ABB RAPID module: LArm

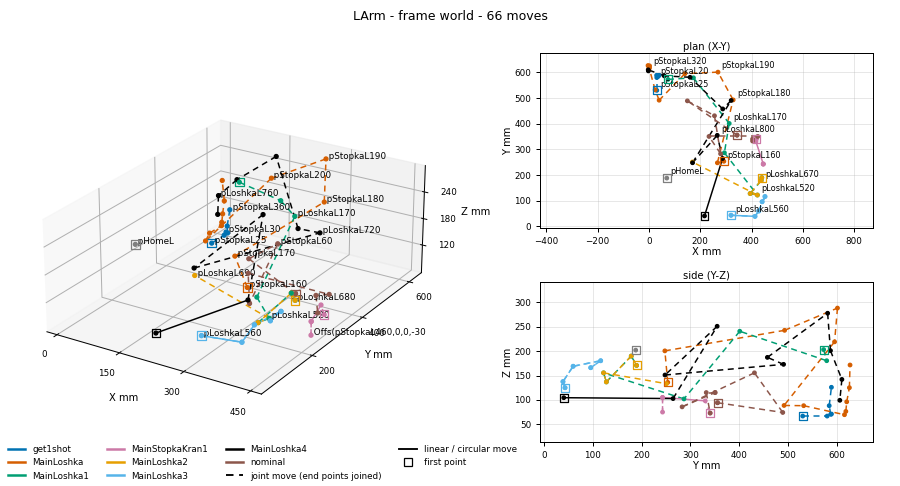
[picture p0: tool path of LArm in frame world, 66 of 71 moves have a stored position in this frame; points joined in program order, loops and branches not executed]
MODULE Barwomen
    PERS num yeetnum:=2;
    PERS num countshots:=1;
    CONST robtarget pHomeL:=[[69.60,187.92,202.03],[0.357643,-0.554439,0.617653,-0.428012],[0,2,-1,5],[91.5197,9E+09,9E+09,9E+09,9E+09,9E+09]];
    CONST robtarget pStopkaL:= [[343.54,355.49,94.31],[0.607961,-0.498613,0.50007,-0.362903],[-1,0,1,4],[102.275,9E+09,9E+09,9E+09,9E+09,9E+09]];
    CONST robtarget pStopkaL10:= [[149.90,489.07,74.39],[0.655337,-0.743509,-0.128276,0.0356828],[-2,-1,2,4],[-6.84347,9E+09,9E+09,9E+09,9E+09,9E+09]];
    CONST robtarget pStopkaL25:=[[30.70,529.98,67.00],[0.666338,-0.744166,-0.0450194,0.0135852],[-1,0,1,4],[4.49505,9E+09,9E+09,9E+09,9E+09,9E+09]];
    CONST robtarget pStopkaL20:=[[30.70,579.98,67.00],[0.666338,-0.744166,-0.0450194,0.0135852],[-1,0,1,4],[4.49505,9E+09,9E+09,9E+09,9E+09,9E+09]];
    CONST robtarget pStopkaL30:=[[30.06,588.78,71.16],[0.666386,-0.744682,-0.0349029,0.0126364],[-1,0,1,4],[4.83424,9E+09,9E+09,9E+09,9E+09,9E+09]];
    CONST robtarget pStopkaL40:=[[30.71,588.95,147.99],[0.686498,-0.726996,0.00257807,-0.0138272],[-1,0,1,5],[-0.204158,9E+09,9E+09,9E+09,9E+09,9E+09]];
    CONST robtarget pStopkaL50:=[[36.78,501.76,153.06],[0.691746,-0.722049,-0.00012744,0.0115038],[-2,0,1,5],[0.0122464,9E+09,9E+09,9E+09,9E+09,9E+09]];
    CONST robtarget pStopkaL60:=[[255.51,431.06,155.58],[0.531694,-0.613357,0.446417,-0.376572],[0,0,1,4],[90.6069,9E+09,9E+09,9E+09,9E+09,9E+09]];
    CONST robtarget pStopkaL70:=[[413.58,330.88,124.32],[0.439492,-0.516452,0.565655,-0.469209],[-1,0,1,4],[120.831,9E+09,9E+09,9E+09,9E+09,9E+09]];
    CONST robtarget pStopkaL90:=[[410.42,334.28,75.42],[0.42637,-0.518144,0.569088,-0.475263],[-1,0,1,4],[118.859,9E+09,9E+09,9E+09,9E+09,9E+09]];
    CONST robtarget pStopkaL100:=[[400.90,338.32,56.69],[0.459651,-0.526008,0.506037,-0.505928],[-1,0,1,4],[119.688,9E+09,9E+09,9E+09,9E+09,9E+09]];
    CONST robtarget pStopkaL110:=[[435.71,243.69,57.40],[0.320976,-0.373543,0.616366,-0.614437],[-1,0,1,4],[141.804,9E+09,9E+09,9E+09,9E+09,9E+09]];
    CONST robtarget pLoshkaL:=[[146.42,414.73,111.00],[0.205105,-0.470911,0.783251,-0.350276],[0,0,0,4],[105.734,9E+09,9E+09,9E+09,9E+09,9E+09]];
    CONST robtarget pLoshkaL40:=[[260.01,572.72,128.57],[0.738375,-0.646351,0.162746,-0.102695],[-1,0,1,4],[26.4369,9E+09,9E+09,9E+09,9E+09,9E+09]];
    CONST robtarget pLoshkaL50:=[[213.98,500.37,132.17],[0.737707,-0.674866,-0.0131158,0.0131439],[-2,0,1,4],[-1.97164,9E+09,9E+09,9E+09,9E+09,9E+09]];
    CONST robtarget pLoshkaL60:=[[94.37,610.04,87.57],[0.723931,-0.683979,-0.0724621,0.0533385],[-1,0,1,4],[-14.2716,9E+09,9E+09,9E+09,9E+09,9E+09]];
    CONST robtarget pLoshkaL70:=[[108.60,590.72,119.23],[0.659052,-0.723466,-0.123201,0.164524],[-1,1,0,5],[16.7664,9E+09,9E+09,9E+09,9E+09,9E+09]];
	CONST robtarget pLoshkaL80:=[[106.05,589.26,170.00],[0.690751,-0.683569,-0.13741,0.191612],[-1,1,0,5],[18.5086,9E+09,9E+09,9E+09,9E+09,9E+09]];
	CONST robtarget pLoshkaL90:=[[99.01,614.59,72.53],[0.67822,-0.729551,-0.0723223,0.0504203],[-1,0,1,4],[-12.518,9E+09,9E+09,9E+09,9E+09,9E+09]];
	CONST robtarget pLoshkaL100:=[[96.19,619.68,93.67],[0.69417,-0.714195,-0.0716613,0.0540104],[-1,0,1,4],[-12.6324,9E+09,9E+09,9E+09,9E+09,9E+09]];
	CONST robtarget pLoshkaL110:=[[99.33,623.54,126.41],[0.757467,-0.648361,-0.0571086,0.0510903],[-1,0,1,4],[-12.6989,9E+09,9E+09,9E+09,9E+09,9E+09]];
	CONST robtarget pLoshkaL120:=[[102.35,603.85,74.33],[0.688053,-0.722838,-0.061305,0.0181653],[-1,0,1,4],[-2.10312,9E+09,9E+09,9E+09,9E+09,9E+09]];
	CONST robtarget pLoshkaL130:=[[112.25,617.73,219.30],[0.80161,-0.596095,-0.0447694,0.00934145],[-1,0,1,4],[-1.00592,9E+09,9E+09,9E+09,9E+09,9E+09]];
	CONST robtarget pLoshkaL140:=[[102.80,608.46,75.78],[0.659248,-0.751754,0.00802967,0.013955],[-1,1,0,4],[-14.6504,9E+09,9E+09,9E+09,9E+09,9E+09]];
	CONST robtarget pStopkaL120:=[[254.59,246.36,160.32],[0.219426,-0.429811,0.719191,-0.499879],[0,2,2,5],[121.393,9E+09,9E+09,9E+09,9E+09,9E+09]];
	CONST robtarget pStopkaL130:=[[208.93,557.30,130.95],[0.677855,-0.732756,-0.0595602,-0.00574711],[-2,3,2,4],[6.35853,9E+09,9E+09,9E+09,9E+09,9E+09]];
	CONST robtarget pStopkaL140:=[[4.38,580.51,84.61],[0.654697,-0.73583,-0.151597,0.0833299],[-1,3,2,5],[-28.9626,9E+09,9E+09,9E+09,9E+09,9E+09]];
	CONST robtarget pStopkaL150:=[[-4.39,620.46,66.05],[0.629943,-0.766063,-0.0798046,0.0997524],[-1,3,2,5],[-30.0775,9E+09,9E+09,9E+09,9E+09,9E+09]];
	CONST robtarget pStopkaL160:=[[292.20,253.51,136.05],[0.329261,-0.370384,0.615322,-0.61301],[0,0,1,4],[124.476,9E+09,9E+09,9E+09,9E+09,9E+09]];
	CONST robtarget pStopkaL170:=[[266.91,247.56,200.56],[0.24886,-0.35748,0.711837,-0.550967],[0,2,3,5],[124.928,9E+09,9E+09,9E+09,9E+09,9E+09]];
	CONST robtarget pStopkaL180:=[[328.40,492.79,242.62],[0.451076,-0.603871,0.576884,-0.314762],[0,2,3,5],[122.987,9E+09,9E+09,9E+09,9E+09,9E+09]];
	CONST robtarget pStopkaL190:=[[269.25,601.13,288.22],[0.801438,-0.576644,-0.0171076,-0.157753],[-1,2,3,5],[22.6915,9E+09,9E+09,9E+09,9E+09,9E+09]];
	CONST robtarget pStopkaL200:=[[140.33,595.16,219.06],[0.75034,-0.655298,-0.068013,0.0543001],[-1,3,3,4],[-2.76391,9E+09,9E+09,9E+09,9E+09,9E+09]];
	CONST robtarget pStopkaL210:=[[12.06,558.03,68.42],[0.640559,-0.739104,-0.1798,0.105267],[-1,2,3,5],[-28.9595,9E+09,9E+09,9E+09,9E+09,9E+09]];
	CONST robtarget pStopkaL220:=[[-2.76,615.20,65.37],[0.627389,-0.758645,-0.138201,0.108357],[-1,3,3,5],[-30.1149,9E+09,9E+09,9E+09,9E+09,9E+09]];
	CONST robtarget pStopkaL230:=[[39.82,491.70,88.73],[0.636114,-0.700358,-0.270169,0.178511],[-2,3,2,4],[-26.5779,9E+09,9E+09,9E+09,9E+09,9E+09]];
	CONST robtarget pStopkaL240:=[[-3.07,608.90,77.17],[0.614365,-0.75743,-0.184586,0.121582],[-1,3,2,5],[-40.2313,9E+09,9E+09,9E+09,9E+09,9E+09]];
	CONST robtarget pStopkaL250:=[[14.08,589.24,87.11],[0.661665,-0.715431,-0.190831,0.118075],[-1,2,-1,5],[-32.2807,9E+09,9E+09,9E+09,9E+09,9E+09]];
	CONST robtarget pStopkaL260:=[[24.16,531.90,88.27],[0.0507054,0.151089,-0.732274,-0.6621],[-1,1,2,5],[-12.6428,9E+09,9E+09,9E+09,9E+09,9E+09]];
	CONST robtarget pStopkaL270:=[[1.33,615.48,69.80],[0.0553407,0.031398,-0.773584,-0.630491],[-1,1,2,4],[-15.0131,9E+09,9E+09,9E+09,9E+09,9E+09]];
	CONST robtarget pStopkaL280:=[[438.60,237.01,70.71],[0.40644,-0.449696,0.548442,-0.576013],[-1,-1,1,4],[146.164,9E+09,9E+09,9E+09,9E+09,9E+09]];
	CONST robtarget pStopkaL290:=[[437.08,242.90,61.40],[0.398327,-0.468707,0.553005,-0.561992],[-1,-1,1,4],[146.104,9E+09,9E+09,9E+09,9E+09,9E+09]];
	CONST robtarget pStopkaL300:=[[-1.35,616.33,70.52],[0.051622,0.0562498,-0.768706,-0.635029],[-1,1,1,5],[6.92965,9E+09,9E+09,9E+09,9E+09,9E+09]];
	CONST robtarget pStopkaL310:=[[0.35,618.29,76.60],[0.0439867,0.0393509,-0.776869,-0.62689],[-1,1,2,4],[-12.4484,9E+09,9E+09,9E+09,9E+09,9E+09]];
	CONST robtarget pStopkaL320:=[[1.52,620.05,96.24],[0.0584018,0.0456965,-0.758439,-0.647512],[-1,1,2,4],[-11.7749,9E+09,9E+09,9E+09,9E+09,9E+09]];
	CONST robtarget pStopkaL330:=[[2.44,625.54,125.12],[0.0668325,0.0457456,-0.734888,-0.673335],[-1,1,2,4],[-11.8794,9E+09,9E+09,9E+09,9E+09,9E+09]];
	CONST robtarget pStopkaL340:=[[-3.52,626.86,171.60],[0.0964834,0.0646992,-0.690576,-0.71387],[-1,1,2,5],[-12.0184,9E+09,9E+09,9E+09,9E+09,9E+09]];
	CONST robtarget pStopkaL80:=[[34.97,587.32,70.63],[0.642788,-0.765376,-0.0129053,0.0292597],[-1,0,1,4],[5.58064,9E+09,9E+09,9E+09,9E+09,9E+09]];
	CONST robtarget pStopkaL350:=[[35.87,584.20,88.27],[0.584467,-0.810973,-0.0153762,0.0220062],[-1,0,1,5],[2.4595,9E+09,9E+09,9E+09,9E+09,9E+09]];
	CONST robtarget pStopkaL360:=[[39.83,588.72,125.94],[0.600543,-0.798875,0.00263761,0.033776],[-1,0,1,5],[1.01816,9E+09,9E+09,9E+09,9E+09,9E+09]];
	CONST robtarget pStopkaL370:=[[423.02,272.97,138.62],[0.497199,0.348722,0.701396,0.373136],[-1,0,2,5],[97.7673,9E+09,9E+09,9E+09,9E+09,9E+09]];
	CONST robtarget pLoshkaL150:=[[74.06,572.76,203.23],[0.127389,0.0200223,-0.660743,-0.739453],[-1,1,2,4],[-17.6646,9E+09,9E+09,9E+09,9E+09,9E+09]];
	CONST robtarget pLoshkaL160:=[[173.49,579.07,180.39],[0.333717,-0.619742,-0.30608,-0.640989],[-1,1,2,5],[80.344,9E+09,9E+09,9E+09,9E+09,9E+09]];
	CONST robtarget pLoshkaL170:=[[313.02,401.00,240.73],[0.75673,-0.320396,0.513231,-0.24759],[-1,2,-1,5],[96.5222,9E+09,9E+09,9E+09,9E+09,9E+09]];
	CONST robtarget pLoshkaL180:=[[306.51,220.57,211.33],[0.761564,-0.20481,0.469899,-0.39657],[-1,2,0,5],[110.246,9E+09,9E+09,9E+09,9E+09,9E+09]];
	CONST robtarget pLoshkaL190:=[[383.36,177.66,210.94],[0.724976,-0.220589,0.394554,-0.51969],[-1,2,-1,5],[108.367,9E+09,9E+09,9E+09,9E+09,9E+09]];
	CONST robtarget pLoshkaL200:=[[421.93,210.16,161.75],[0.622169,-0.40055,0.454591,-0.495794],[-1,2,-1,5],[107.286,9E+09,9E+09,9E+09,9E+09,9E+09]];
	CONST robtarget pLoshkaL210:=[[381.08,197.44,210.52],[0.735266,-0.426091,0.316311,-0.421637],[-1,1,0,5],[113.423,9E+09,9E+09,9E+09,9E+09,9E+09]];
	CONST robtarget pLoshkaL220:=[[409.44,209.14,193.34],[0.689351,-0.445905,0.384231,-0.422291],[-1,1,0,5],[110.848,9E+09,9E+09,9E+09,9E+09,9E+09]];
	CONST robtarget pLoshkaL230:=[[434.76,220.01,164.41],[0.616775,-0.472773,0.461444,-0.427954],[-1,1,0,5],[108.199,9E+09,9E+09,9E+09,9E+09,9E+09]];
	CONST robtarget pLoshkaL240:=[[317.22,283.65,170.47],[0.640998,-0.146442,0.747547,0.0940749],[0,1,1,5],[109.871,9E+09,9E+09,9E+09,9E+09,9E+09]];
	CONST robtarget pLoshkaL250:=[[418.67,130.38,165.04],[0.634652,-0.100699,0.730731,-0.230453],[-1,1,1,5],[112.705,9E+09,9E+09,9E+09,9E+09,9E+09]];
	CONST robtarget pLoshkaL260:=[[432.52,161.66,186.76],[0.583769,-0.268113,0.679713,-0.354006],[-1,1,0,5],[110.556,9E+09,9E+09,9E+09,9E+09,9E+09]];
	CONST robtarget pLoshkaL270:=[[429.00,215.51,153.40],[0.530561,-0.454209,0.61183,-0.371298],[-1,1,0,5],[109.073,9E+09,9E+09,9E+09,9E+09,9E+09]];
	CONST robtarget pLoshkaL280:=[[255.79,417.68,226.75],[0.725186,0.00109822,0.686472,-0.0534826],[0,2,-1,5],[83.0807,9E+09,9E+09,9E+09,9E+09,9E+09]];
	CONST robtarget pLoshkaL290:=[[289.16,236.70,183.45],[0.674629,-0.106946,0.686871,-0.248289],[0,2,0,5],[105.927,9E+09,9E+09,9E+09,9E+09,9E+09]];
	CONST robtarget pLoshkaL300:=[[389.96,136.16,152.69],[0.701811,-0.0448875,0.634194,-0.321317],[-1,2,0,5],[111.143,9E+09,9E+09,9E+09,9E+09,9E+09]];
	CONST robtarget pLoshkaL310:=[[433.03,205.08,156.97],[0.560134,-0.389099,0.585763,-0.437874],[-1,2,-1,5],[108.185,9E+09,9E+09,9E+09,9E+09,9E+09]];
	CONST robtarget pLoshkaL320:=[[321.63,255.70,162.17],[0.615082,-0.251421,0.747187,-0.0131705],[0,1,1,5],[114.69,9E+09,9E+09,9E+09,9E+09,9E+09]];
	CONST robtarget pLoshkaL330:=[[422.99,136.85,170.78],[0.663877,-0.282999,0.684499,-0.103155],[-1,1,1,5],[117.899,9E+09,9E+09,9E+09,9E+09,9E+09]];
	CONST robtarget pLoshkaL340:=[[415.82,205.67,184.27],[0.627658,-0.590253,0.406647,-0.303785],[-1,1,0,5],[114.688,9E+09,9E+09,9E+09,9E+09,9E+09]];
	CONST robtarget pLoshkaL350:=[[427.25,218.21,157.00],[0.565395,-0.627354,0.446388,-0.295792],[-1,1,0,5],[112.591,9E+09,9E+09,9E+09,9E+09,9E+09]];
	CONST robtarget pLoshkaL360:=[[281.30,379.43,103.44],[0.105219,-0.862829,-0.0249149,-0.493796],[0,1,2,5],[97.9634,9E+09,9E+09,9E+09,9E+09,9E+09]];
	CONST robtarget pLoshkaL370:=[[294.22,286.68,102.12],[0.529015,-0.117018,0.838074,-0.0638862],[0,0,-2,4],[105.801,9E+09,9E+09,9E+09,9E+09,9E+09]];
	CONST robtarget pLoshkaL380:=[[354.81,135.82,123.45],[0.640211,0.0205258,0.74832,-0.172411],[-1,0,-2,4],[114.811,9E+09,9E+09,9E+09,9E+09,9E+09]];
	CONST robtarget pLoshkaL390:=[[395.62,127.40,133.97],[0.636248,-0.0240691,0.741395,-0.211997],[-1,0,-2,4],[113.914,9E+09,9E+09,9E+09,9E+09,9E+09]];
	CONST robtarget pLoshkaL400:=[[409.39,125.22,135.99],[0.542603,-0.00983826,0.814196,-0.206326],[-1,0,-2,5],[111.62,9E+09,9E+09,9E+09,9E+09,9E+09]];
	CONST robtarget pLoshkaL410:=[[422.57,130.61,142.57],[0.525991,-0.0373933,0.804774,-0.272531],[-1,0,-2,5],[118.167,9E+09,9E+09,9E+09,9E+09,9E+09]];
	CONST robtarget pLoshkaL420:=[[432.11,181.18,170.00],[0.59696,-0.314212,0.612857,-0.41148],[-1,-1,-2,4],[119.634,9E+09,9E+09,9E+09,9E+09,9E+09]];
	CONST robtarget pLoshkaL430:=[[423.76,206.02,154.80],[0.605126,-0.38377,0.529881,-0.453618],[-1,-1,-2,4],[119.97,9E+09,9E+09,9E+09,9E+09,9E+09]];
	CONST robtarget pStopkaL380:=[[279.44,282.90,85.87],[0.464873,-0.562779,0.539692,-0.419411],[0,-1,1,4],[123.903,9E+09,9E+09,9E+09,9E+09,9E+09]];
	CONST robtarget pStopkaL390:=[[215.92,370.13,114.84],[0.542845,-0.586286,0.441093,-0.408687],[0,-1,1,4],[127.367,9E+09,9E+09,9E+09,9E+09,9E+09]];
	CONST robtarget pStopkaL400:=[[234.21,350.40,115.15],[0.542694,-0.584981,0.44227,-0.409484],[0,-1,1,4],[127.384,9E+09,9E+09,9E+09,9E+09,9E+09]];
    CONST robtarget pStopkaL410:=[[404.22,350.38,115.15],[0.542685,-0.584976,0.442274,-0.4095],[-1,-1,1,4],[127.384,9E+09,9E+09,9E+09,9E+09,9E+09]];
    CONST robtarget pStopkaL420:=[[404.23,340.37,115.15],[0.542677,-0.58497,0.442279,-0.409513],[-1,-1,1,4],[127.384,9E+09,9E+09,9E+09,9E+09,9E+09]];
    CONST robtarget pStopkaL430:=[[404.23,340.36,73.15],[0.542669,-0.584964,0.442284,-0.409527],[-1,-1,1,4],[127.384,9E+09,9E+09,9E+09,9E+09,9E+09]];
    CONST robtarget pStopkaL440:=[[417.24,340.35,73.15],[0.542661,-0.584958,0.442289,-0.409541],[-1,-1,1,4],[127.384,9E+09,9E+09,9E+09,9E+09,9E+09]];
    CONST robtarget pStopkaL450:=[[445.71,242.85,105.14],[0.554038,-0.578654,0.404196,-0.441392],[-1,-1,2,4],[134.835,9E+09,9E+09,9E+09,9E+09,9E+09]];
    CONST robtarget pStopkaL460:=[[445.71,242.84,105.14],[0.55403,-0.57865,0.4042,-0.441404],[-1,-1,2,4],[134.835,9E+09,9E+09,9E+09,9E+09,9E+09]];
    CONST robtarget pStopkaL470:=[[445.71,242.83,75.14],[0.554023,-0.578644,0.404205,-0.441414],[-1,-1,2,4],[134.835,9E+09,9E+09,9E+09,9E+09,9E+09]];
    CONST robtarget pLoshkaL440:=[[436.61,201.35,158.18],[0.480333,-0.407272,0.617894,-0.470763],[-1,-1,-3,4],[117.231,9E+09,9E+09,9E+09,9E+09,9E+09]];
    CONST robtarget pLoshkaL450:=[[442.08,206.24,178.64],[0.462949,-0.41361,0.619401,-0.48057],[-1,-1,-2,4],[116.494,9E+09,9E+09,9E+09,9E+09,9E+09]];
    CONST robtarget pLoshkaL460:=[[438.64,185.76,191.95],[0.483869,-0.330718,0.672419,-0.45205],[-1,-1,-2,5],[116.918,9E+09,9E+09,9E+09,9E+09,9E+09]];
    CONST robtarget pLoshkaL470:=[[441.68,180.53,213.10],[0.503033,-0.320898,0.651608,-0.46839],[-1,-1,-2,5],[117.275,9E+09,9E+09,9E+09,9E+09,9E+09]];
    CONST robtarget pLoshkaL480:=[[419.78,172.39,165.82],[0.50331,-0.09878,0.812631,-0.276682],[-1,0,-2,5],[116.99,9E+09,9E+09,9E+09,9E+09,9E+09]];
    CONST robtarget pLoshkaL490:=[[330.12,200.97,156.56],[0.522475,-0.160719,0.79702,-0.256804],[0,0,-2,4],[117.927,9E+09,9E+09,9E+09,9E+09,9E+09]];
    CONST robtarget pLoshkaL500:=[[237.41,251.34,109.43],[0.623306,0.0127326,0.773395,-0.114843],[0,0,-2,4],[112.654,9E+09,9E+09,9E+09,9E+09,9E+09]];
    CONST robtarget pLoshkaL510:=[[442.48,135.74,167.58],[0.558188,-0.134718,0.723644,-0.382905],[-1,-1,-2,4],[127.982,9E+09,9E+09,9E+09,9E+09,9E+09]];
    CONST robtarget pLoshkaL520:=[[422.90,122.02,155.52],[0.551222,0.0407261,0.768447,-0.322467],[-1,0,-2,4],[137.837,9E+09,9E+09,9E+09,9E+09,9E+09]];
    CONST robtarget pLoshkaL530:=[[441.36,146.50,170.40],[0.543256,-0.16596,0.704956,-0.424696],[-1,-1,-2,4],[137.81,9E+09,9E+09,9E+09,9E+09,9E+09]];
    CONST robtarget pLoshkaL540:=[[431.40,196.95,172.43],[0.570337,-0.284228,0.581124,-0.506186],[-1,-1,-3,4],[138.317,9E+09,9E+09,9E+09,9E+09,9E+09]];
    CONST robtarget pLoshkaL550:=[[441.69,207.71,153.91],[0.540425,-0.375422,0.560952,-0.502327],[-1,-1,-3,4],[138.493,9E+09,9E+09,9E+09,9E+09,9E+09]];
    CONST robtarget pLoshkaL560:=[[320.01,43.09,125.04],[0.656848,0.181676,0.666032,-0.303227],[-1,0,-2,4],[125.934,9E+09,9E+09,9E+09,9E+09,9E+09]];
    CONST robtarget pLoshkaL570:=[[413.50,38.86,137.56],[0.64945,0.116654,0.69766,-0.279063],[-1,0,-2,4],[122.529,9E+09,9E+09,9E+09,9E+09,9E+09]];
    CONST robtarget pLoshkaL580:=[[428.04,59.72,169.02],[0.623701,-0.0735723,0.640429,-0.44208],[-1,0,-2,4],[121.294,9E+09,9E+09,9E+09,9E+09,9E+09]];
    CONST robtarget pLoshkaL590:=[[452.43,116.13,180.32],[0.556864,-0.327476,0.531563,-0.547817],[-1,0,-3,4],[120.131,9E+09,9E+09,9E+09,9E+09,9E+09]];
    CONST robtarget pLoshkaL600:=[[441.27,95.75,166.10],[0.594154,-0.22301,0.585847,-0.504015],[-1,0,-3,4],[120.649,9E+09,9E+09,9E+09,9E+09,9E+09]];
    CONST robtarget pCalib:=[[80.69,507.44,67.00],[0.666335,-0.744165,-0.0450548,0.0136173],[-2,0,1,4],[4.49551,9E+09,9E+09,9E+09,9E+09,9E+09]];
    CONST robtarget pLoshkaL610:=[[394.69,127.73,136.94],[0.523705,0.0379416,0.79027,-0.315859],[-1,0,-2,4],[138.35,9E+09,9E+09,9E+09,9E+09,9E+09]];
    CONST robtarget pLoshkaL620:=[[413.12,160.92,196.32],[0.5222,-0.186845,0.68287,-0.475484],[-1,0,-3,4],[137.891,9E+09,9E+09,9E+09,9E+09,9E+09]];
    CONST robtarget pLoshkaL630:=[[431.78,196.82,172.35],[0.499901,-0.349323,0.618102,-0.496007],[-1,-1,-3,4],[137.681,9E+09,9E+09,9E+09,9E+09,9E+09]];
    CONST robtarget pLoshkaL640:=[[402.08,126.31,144.27],[0.173047,0.80248,-0.0154847,0.570825],[-1,2,-2,4],[117.174,9E+09,9E+09,9E+09,9E+09,9E+09]];
    CONST robtarget pLoshkaL650:=[[432.54,158.50,192.59],[0.341162,0.748933,0.223016,0.522467],[-1,2,-3,4],[113.743,9E+09,9E+09,9E+09,9E+09,9E+09]];
    CONST robtarget pLoshkaL660:=[[436.96,190.59,204.87],[0.445322,0.655486,0.347248,0.501443],[-1,1,-3,4],[112.213,9E+09,9E+09,9E+09,9E+09,9E+09]];
    CONST robtarget pLoshkaL670:=[[437.73,178.72,189.87],[0.557027,-0.315306,0.606495,-0.471665],[-1,-1,-2,4],[138.63,9E+09,9E+09,9E+09,9E+09,9E+09]];
    CONST robtarget pLoshkaL680:=[[440.02,189.65,170.79],[0.53203,-0.342362,0.606016,-0.482159],[-1,-1,-2,4],[138.35,9E+09,9E+09,9E+09,9E+09,9E+09]];
    CONST robtarget pLoshkaL690:=[[169.50,250.84,133.34],[0.520043,0.0199626,0.845698,-0.118118],[0,0,-2,4],[104.383,9E+09,9E+09,9E+09,9E+09,9E+09]];
    CONST robtarget pLoshkaL700:=[[314.93,145.15,136.89],[0.66465,0.144156,0.721464,-0.130189],[-1,2,0,5],[120.915,9E+09,9E+09,9E+09,9E+09,9E+09]];
    CONST robtarget pLoshkaL710:=[[170.09,247.87,151.08],[0.631674,0.0466004,0.771386,-0.0614899],[0,2,0,5],[107.07,9E+09,9E+09,9E+09,9E+09,9E+09]];
    CONST robtarget pLoshkaL720:=[[320.68,490.67,172.94],[0.424079,0.178298,0.557136,0.691351],[-1,2,1,5],[69.7446,9E+09,9E+09,9E+09,9E+09,9E+09]];
    CONST robtarget pLoshkaL730:=[[287.81,457.60,187.22],[0.413312,0.37036,0.551339,0.622922],[-1,2,1,5],[83.6966,9E+09,9E+09,9E+09,9E+09,9E+09]];
    CONST robtarget pLoshkaL740:=[[160.36,580.97,277.61],[0.0503744,0.12748,0.486421,0.862905],[-1,2,1,5],[29.8157,9E+09,9E+09,9E+09,9E+09,9E+09]];
    CONST robtarget pLoshkaL750:=[[59.49,586.76,201.05],[0.0518925,0.110024,-0.545861,-0.828998],[-1,2,1,5],[-0.225623,9E+09,9E+09,9E+09,9E+09,9E+09]];
    CONST robtarget pLoshkaL760:=[[-2.69,610.17,142.05],[0.00451034,0.0888736,-0.829709,-0.551057],[-1,2,1,4],[-22.5532,9E+09,9E+09,9E+09,9E+09,9E+09]];
    CONST robtarget pLoshkaL770:=[[-2.20,605.95,99.33],[0.0503534,0.082125,-0.847594,-0.521828],[-1,2,1,4],[-17.0162,9E+09,9E+09,9E+09,9E+09,9E+09]];
    CONST robtarget pLoshkaL780:=[[216.66,40.49,104.62],[0.615541,0.302515,0.663302,-0.299374],[-1,0,-2,4],[124.852,9E+09,9E+09,9E+09,9E+09,9E+09]];
    CONST robtarget pLoshkaL790:=[[287.08,264.39,102.85],[0.606655,0.104461,0.783718,-0.0827291],[0,0,-2,4],[112.694,9E+09,9E+09,9E+09,9E+09,9E+09]];
    CONST robtarget pLoshkaL800:=[[266.45,354.68,250.93],[0.0713052,0.637415,0.0090863,0.767161],[0,0,0,4],[103.37,9E+09,9E+09,9E+09,9E+09,9E+09]];

    PROC get1shot()
         MoveJ pStopkaL25, v50, z0, GripperL;
         MoveJ pStopkaL20, v50, z0, GripperL;
         MoveJ pStopkaL30, v50, z0, GripperL;
         WaitTime 1;
         g_GripIn;
         MoveJ pStopkaL80, v50, z0, GripperL;
         MoveJ pStopkaL350, v50, z0, GripperL;
         MoveJ pStopkaL360, v50, z0, GripperL;
    ENDPROC
    PROC MainLoshka()
        MoveJ pStopkaL160, v50, z0, GripperL;
         MoveJ pStopkaL170, v150, z0, GripperL;
         MoveJ pStopkaL180, v150, z0, GripperL;
         MoveJ pStopkaL190, v150, z0, GripperL;
         MoveJ pStopkaL200, v150, z0, GripperL;
         MoveJ pStopkaL230, v150, z0, GripperL;
         MoveJ pStopkaL260, v150, z0, GripperL;
         MoveJ pStopkaL270, v150, z0, GripperL;
         WaitTime 2;
         g_GripIn;
         WaitTime 1;
         MoveJ pStopkaL310, v100,fine , GripperL;
         MoveJ pStopkaL320, v100, fine, GripperL;
         MoveJ pStopkaL330, v100, fine, GripperL;
         MoveJ pStopkaL340, v100, fine, GripperL;
    ENDPROC
    PROC MainLoshka1()
         MoveJ pLoshkaL150, v100, z0, GripperL;
         MoveJ pLoshkaL160, v100, z0, GripperL;
         MoveJ pLoshkaL170, v100, z0, GripperL;
         MoveJ pLoshkaL370, v100, z0, GripperL;
         MoveJ pLoshkaL520, v100, z0, GripperL;
         MoveJ pLoshkaL610, v100, z0, GripperL;
         MoveJ pLoshkaL670, v100, z0, GripperL;
         MoveJ pLoshkaL680, v100, z0, GripperL;
         WaitTime 2;
         SetDo custom_do_0,0;
         WaitDo custom_do_0,2;
!         WaitTime 10;
    ENDPROC
    PROC MainStopkaKran1()
         MoveJ Offs( pStopkaL430,15,0,0), v50, fine, GripperL;
!         MoveJ pStopkaL100, v150, fine, GripperL;
         g_GripIn;
         MoveJ Offs( pStopkaL440,0,-10,25), v50, fine, GripperL;
         MoveL pStopkaL450, v50, fine, GripperL;
         MoveJ Offs(pStopkaL460,0,0,-30), v50, fine, GripperL;
         WaitTime 1;
!         MoveJ pStopkaL280, v50, fine, GripperL;
!         MoveJ pStopkaL290, v50, fine, GripperL;
         g_GripOut;
         WaitTime 1;
!         MoveJ  pStopkaL470, v50, fine, GripperL;
         MoveJ Offs(pStopkaL470,0,0,30), v50, fine, GripperL;
    ENDPROC
    PROC MainLoshka2()
        MoveJ pLoshkaL680, v100, z0, GripperL;
        MoveJ pLoshkaL670, v100, z0, GripperL;
        MoveJ pLoshkaL610, v100, z0, GripperL;
        MoveJ pLoshkaL520, v100, z0, GripperL;
        MoveJ pLoshkaL690, v100, z0, GripperL;
        WaitDO custom_do_0,0;
    ENDPROC

    PROC MainLoshka3()
        g_GripIn;
        MoveL pLoshkaL560, v150, fine, GripperL;
        MoveJ pLoshkaL570, v150, fine, GripperL;
        MoveJ pLoshkaL580, v150, fine, GripperL;
        MoveJ pLoshkaL590, v150, fine, GripperL;
        MoveJ pLoshkaL600, v150, fine, GripperL;
        SetDo  custom_DO_0,1;
	WaitDO custom_do_0,0;
	MoveJ pLoshkaL600, v150, fine, GripperL;
	MoveJ pLoshkaL590, v150, fine, GripperL;
	MoveJ pLoshkaL580, v150, fine, GripperL;
	MoveJ pLoshkaL570, v150, fine, GripperL;
	MoveL pLoshkaL560, v150, fine, GripperL;
    ENDPROC
    PROC MainLoshka4()
        MoveL pLoshkaL780, v150, z0, GripperL;
        MoveL pLoshkaL790, v150, z0, GripperL;
        MoveJ pLoshkaL800, v150, z0, GripperL;
        MoveJ pLoshkaL710, v150, z0, GripperL;
        MoveJ pLoshkaL720, v150, z0, GripperL;
        MoveJ pLoshkaL730, v150, z0, GripperL;
        MoveJ pLoshkaL740, v150, z0, GripperL;
        MoveJ pLoshkaL750, v150, z0, GripperL;
        MoveJ pLoshkaL760, v150, fine, GripperL;
        MoveJ pLoshkaL770, v150, fine, GripperL;
        g_GripOut;
        SetDo  custom_DO_0,1;

    ENDPROC

    PROC GetNot1Shot(num off)

         MoveJ Offs(pCalib,off,0,0), v150, z0, GripperL;
         MoveJ Offs(pStopkaL20,off,0,0), v150, z0, GripperL;
         MoveJ Offs(pStopkaL30,off,0,0), v150, z0, GripperL;
         WaitTime 1;
         g_GripIn;
         MoveJ Offs(pStopkaL40,off,0,0), v150, z0, GripperL;
         MoveJ Offs(pStopkaL50,off,0,0), v150, z0, GripperL;

    ENDPROC

    PROC nominal()
        MoveJ pStopkaL, v200, z5, GripperL;
        IF yeetnum>6 or yeetnum<1 or countshots>6 THEN
            TPReadFK reg2, "Check shots", "All Clear", "Abort", stEmpty, stEmpty, stEmpty;
            IF reg2=1 THEN
                 yeetnum:=1;
                 countshots:=0;
            ELSE
                MoveJ pStopkaL, v150, z5, GripperL;
                main;
            ENDIF
        ENDIF
         MoveJ pStopkaL10, v150, z0, GripperL;
         !WaitTime 100;
         TEST yeetnum
            CASE 1: get1shot;
            CASE 2: GetNot1Shot(50*(yeetnum-1));
            CASE 3: GetNot1Shot(50*(yeetnum-1));
            CASE 4: GetNot1Shot(50*(yeetnum-1));
            CASE 5: GetNot1Shot(50*(yeetnum-1));
            CASE 6: GetNot1Shot(50*(yeetnum-1));
        ENDTEST
         yeetnum:=yeetnum+1;
         countshots:=countshots+1;
         waittime 1;
         MoveJ pStopkaL60, v150, z0, GripperL;
         MoveJ pStopkaL380, v150, z0, GripperL;
         MoveJ pStopkaL400, v150, z0, GripperL;
         MoveJ Offs(pStopkaL400,190,0,0), v100, z0,GripperL;
         WaitTime 1;
         MoveJ Offs( pStopkaL410,0,-18,0), v50, z0, GripperL;
         WaitTime 1;
         MoveJ Offs (pStopkaL420,0,0,-42), v50, z0, GripperL;
         WaitTime 1;

!        MoveJ pStopkaL90, v50, z0, GripperL;
         WaitTime 2;
         g_SetMaxSpd 5;
         g_GripOut;
         SetDo custom_do_0,0;
         WaitDo custom_do_0,1;
!         MoveJ pStopkaL100, v150, fine, GripperL;
!         g_GripIn;
!         MoveJ pStopkaL280, v50, fine, GripperL;
!         MoveJ pStopkaL290, v50, fine, GripperL;
!         g_GripOut;
!         WaitTime 2;
         !poexal za loshkoi!
         MainStopkaKran1;
         MainLoshka;
!         MainStopkaKran;
         MainLoshka1;
         MainLoshka2;
         MainLoshka3;
         MainLoshka4;
         WaitDO custom_DO_5,0;
!         main;
    ENDPROC




    PROC main()
         !go to stopka!
         SetDO custom_DO_0,1;
         TPErase;
         MoveJ pHomeL, v150, z5, GripperL;
         g_gripout;
         TPReadFK reg1, "Station ready", stEmpty, stEmpty, stEmpty, stEmpty, "Pour the liquid";
         IF reg1=5 THEN
             nominal;
         ENDIF

         !g_SetMaxSpd 4;
         !g_SetForce 5;
         !g_Init;

    ENDPROC
ENDMODULE
